// TIA Portal project "PLC-1200" (V19)

(* hardware
DEVICE "PLC-1200"  S7-1200 Station
   slot 0: "Rack_0"  S7-1200 Rack  Rack  V1.0
   slot 1: "PLC-1200"  CPU 1212C DC/DC/DC  6ES7 212-1AE40-0XB0  V4.6
*)

// ===== PLC "PLC-1200"  CPU 1212C DC/DC/DC =====

TYPE "Crossroad_Input"
   STRUCT
      btnStart : Bool := FALSE;
      btnPause : Bool := FALSE;
      btnStop : Bool := FALSE;
      btnCrosswalk1 : Bool := FALSE;
      btnCrosswalk2 : Bool := FALSE;
   END_STRUCT;
END_TYPE

TYPE "Crossroad_Output"
   STRUCT
      crossroadType : Bool := FALSE;
      trafficLightGreen1 : Bool := FALSE;
      trafficLightsYellow1 : Bool := FALSE;
      trafficLightsRed1 : Bool := FALSE;
      trafficLightGreen2 : Bool := FALSE;
      trafficLightsYellow2 : Bool := FALSE;
      trafficLightsRed2 : Bool := FALSE;
      pedestrianLightGreen1 : Bool := FALSE;
      pedestrianLightRed1 : Bool := FALSE;
      pedestrianLightGreen2 : Bool := FALSE;
      pedestrianLightRed2 : Bool := FALSE;
   END_STRUCT;
END_TYPE

TYPE "Crosswalk_Input"
   STRUCT
      btnStart : Bool := FALSE;
      btnPause : Bool := FALSE;
      btnStop : Bool := FALSE;
      btnCrosswalk1 : Bool := FALSE;
      btnCrosswalk2 : Bool := FALSE;
   END_STRUCT;
END_TYPE

TYPE "Crosswalk_Output"
   STRUCT
      crosswalkType : Bool := FALSE;
      trafficLightGreen1 : Bool := FALSE;
      trafficLightsYellow1 : Bool := FALSE;
      trafficLightsRed1 : Bool := FALSE;
      trafficLightGreen2 : Bool := FALSE;
      trafficLightsYellow2 : Bool := FALSE;
      trafficLightsRed2 : Bool := FALSE;
      pedestrianLightGreen1 : Bool := FALSE;
      pedestrianLightRed1 : Bool := FALSE;
      pedestrianLightGreen2 : Bool := FALSE;
      pedestrianLightRed2 : Bool := FALSE;
   END_STRUCT;
END_TYPE

TYPE "Regulator_Input"
   STRUCT
      switchstate : Bool := FALSE;
      order : Int := 1;
      R1 : Real := 0.0;
      R2 : Real := 0.0;
      C1 : Real := 0.0;
      C2 : Real := 0.0;
      Uin : Real := 0.0;
      Td : Real := 0.0;
      Ts : Real := 0.0;
   END_STRUCT;
END_TYPE

TYPE "Regulator_Output"
   STRUCT
      Uc1 : Real := 0.0;
      Uc2 : Real := 0.0;
      PV : Real := 0.0;
   END_STRUCT;
END_TYPE

TYPE "CarWash_Input"
   STRUCT
      btnEmergencyStop : Bool := FALSE;
      btnStart : Bool := FALSE;
      btnStop : Bool := FALSE;
      ErrorSystem : Bool := FALSE;
      CarPosition : Bool := FALSE;
      ShowerPosition : Bool := FALSE;
      Mode : Int := 0;
   END_STRUCT;
END_TYPE

TYPE "CarWash_Output"
   STRUCT
      Light_green : Bool := FALSE;
      Light_yellow : Bool := FALSE;
      Light_red : Bool := FALSE;
      Door1_Up : Bool := FALSE;
      Door1_Down : Bool := FALSE;
      Door2_Up : Bool := FALSE;
      CarWashDoor2_Down : Bool := FALSE;
      ChemicalsFront : Bool := FALSE;
      ChemicalsSides : Bool := FALSE;
      ChemicalsBack : Bool := FALSE;
      Prewash : Bool := FALSE;
      Water : Bool := FALSE;
      Wax : Bool := FALSE;
      Dry : Bool := FALSE;
      Brushes : Bool := FALSE;
      Soap : Bool := FALSE;
      TimeDoorMovement : Int := 0;
      MEMDoor : Bool := FALSE;
      MEMDoorMovement : Bool := FALSE;
      MEMDoorClosingTrig : Bool := FALSE;
   END_STRUCT;
END_TYPE

TYPE "WashingMachine_Input"
   STRUCT
      btnEmergencyStop : Bool := FALSE;
      btnMachine : Bool := FALSE;
      btnStop : Bool := FALSE;
      ErrorSystem : Bool := FALSE;
      Mode : Int := 0;
   END_STRUCT;
END_TYPE

TYPE "WashingMachine_Output"
   STRUCT
      Light_green : Bool := FALSE;
      Light_yellow : Bool := FALSE;
      Light_red : Bool := FALSE;
      DoorClosed : Bool := FALSE;
      PreWash : Bool := FALSE;
      Water : Bool := FALSE;
      Wax : Bool := FALSE;
      Dry : Bool := FALSE;
      Brushes : Bool := FALSE;
      Soap : Bool := FALSE;
      ActiveFoam : Bool := FALSE;
   END_STRUCT;
END_TYPE

TYPE "CarLight_Input"
   STRUCT
      btnStart : Bool := FALSE;
      btnReset : Bool := FALSE;
      markerLight : Bool := FALSE;
      brakeLight : Bool := FALSE;
      turnLight : Bool := FALSE;
   END_STRUCT;
END_TYPE

TYPE "CarLight_Output"
   STRUCT
      sensorPosition : Bool := FALSE;
      sensorConnectorConnected : Bool := FALSE;
      done : Bool := FALSE;
   END_STRUCT;
END_TYPE

DATA_BLOCK "DB_ProcessData"   // DB1
{ S7_Optimized_Access := 'TRUE' }
VERSION : 0.1
   VAR
      crossroad_input : "Crossroad_Input";
      crossroad_output : "Crossroad_Output";
      crosswalk_input : "Crosswalk_Input";
      crosswalk_output : "Crosswalk_Output";
      regulator_input : "Regulator_Input";
      regulator_output : "Regulator_Output";
      carwash_input : "CarWash_Input";
      carwash_output : "CarWash_Output";
      washingmachine_input : "WashingMachine_Input";
      washingmachine_output : "WashingMachine_Output";
      carlight_input : "CarLight_Input";
      carlight_output : "CarLight_Output";
   END_VAR
BEGIN
END_DATA_BLOCK

ORGANIZATION_BLOCK "Main"   // OB1, LAD, ProgramCycle
TITLE = "Main Program Sweep (Cycle)"
{ S7_Optimized_Access := 'TRUE' }
VERSION : 0.1
   VAR_INPUT
      Initial_Call : Bool;   // Initial call of this OB
      Remanence : Bool;   // =True, if remanent data are available
   END_VAR
BEGIN
END_ORGANIZATION_BLOCK